Staubli VAL3: ReadMatchPreset.pgx

public program ReadMatchPreset(string x_sFileName (dimensions=1), string x_sPresetName (dimensions=1), bool& x_bRes (dimensions=1))
  local num l_nNum[3]
  local string l_sBuff
  local string l_sFileName
begin

  //读取动作文本
  //动作一共是200项，每项12个动作，每个动作一共是一个值
  //


  //参数初始化
  x_bRes=false
  l_sFileName=x_sFileName

  //判断文件是否存在
  if !$fileExists(l_sFileName)
    return
  endIf

  //关闭所有文件
  call FileDir:CloseAllFile()

  //文件是否可以打开
  nFileID=$fileOpen(l_sFileName,"r")
  if nFileID<0 or nFileID>9
    return
  endIf

  //对于原有值进行初始化
  for l_nNum[0]=0 to 200
    for l_nNum[1]=0 to 4
      nMatchPreset[l_nNum[0],l_nNum[1]]=0
    endFor
  endFor


  l_nNum[0]=l_nNum[1]=l_nNum[2]=0


  //读取每行并解析
  if $fileGet(nFileID,l_sBuff,1)!=1 or find(l_sBuff,"PRESET="+x_sPresetName)<0
    return
  endIf

  while $fileGet(nFileID,l_sBuff,1)==1 and l_sBuff!="" and l_nNum[0]<200
    call FileDir:SplitPresetLine(l_sBuff,nMatchPreset,l_nNum[0]+1,x_bRes)
    if !x_bRes
      return
    endIf
    l_nNum[0]=l_nNum[0]+1
  endWhile

  x_bRes=true

  //关闭所有文件
  call FileDir:CloseAllFile()






end
